FUNCTION F_CheckAxisGRT : BOOL
VAR_INPUT
    stMotionStage: ST_MotionStage;
    fQueryValue: LREAL;
END_VAR
VAR
END_VAR

F_CheckAxisGRT := F_CheckAxis(stMotionStage, 2, fQueryValue);

END_FUNCTION

(* stored: Version 1.1.0.1, ProductVersion 3.1.4022.18
   POU F_CheckAxisGRT: Id {731dc843-c335-44d1-b5ac-400491a2bf7a}, SpecialFunc None *)
